// TIA Portal V18 export
FUNCTION_BLOCK "BOOL_DEMUX"   // FB13, LAD
{ S7_Optimized_Access := 'TRUE' }
VERSION : 0.1
// stored: AutoNumber true, IsIECCheckEnabled false, IsRetainMemResEnabled false, MemoryReserve 100, SetENOAutomatically false, UDAEnableTagReadback false
   VAR_INPUT
      State : Int;
      Reset_cmd : Bool;
      Homing_all_axis : Bool;
   END_VAR
   VAR_OUTPUT
      Out1 { ExternalAccessible := 'False'; ExternalVisible := 'False'; ExternalWritable := 'False'} : Bool;
      Out2 { ExternalAccessible := 'False'; ExternalVisible := 'False'; ExternalWritable := 'False'} : Bool;
      Out3 { ExternalAccessible := 'False'; ExternalVisible := 'False'; ExternalWritable := 'False'} : Bool;
      Out4 { ExternalAccessible := 'False'; ExternalVisible := 'False'; ExternalWritable := 'False'} : Bool;
      Out5 { ExternalAccessible := 'False'; ExternalVisible := 'False'; ExternalWritable := 'False'} : Bool;
      Out6 : Int;
   END_VAR
   VAR
      Edge_S_Out1 : Bool;
      Edge_M_Out1 : Bool;
      Edge_S_Out2 : Bool;
      Edge_M_Out2 : Bool;
      Edge_S_Out3 : Bool;
      Edge_M_Out3 : Bool;
      Edge_S_Out4 : Bool;
      Edge_M_Out4 : Bool;
      Edge_S_Out5 : Bool;
      Edge_M_Out5 : Bool;
   END_VAR
   VAR_TEMP   // added for the SCL form of the ladder/FBD networks
      _w1 : Bool;
   END_VAR
BEGIN

REGION Network 1
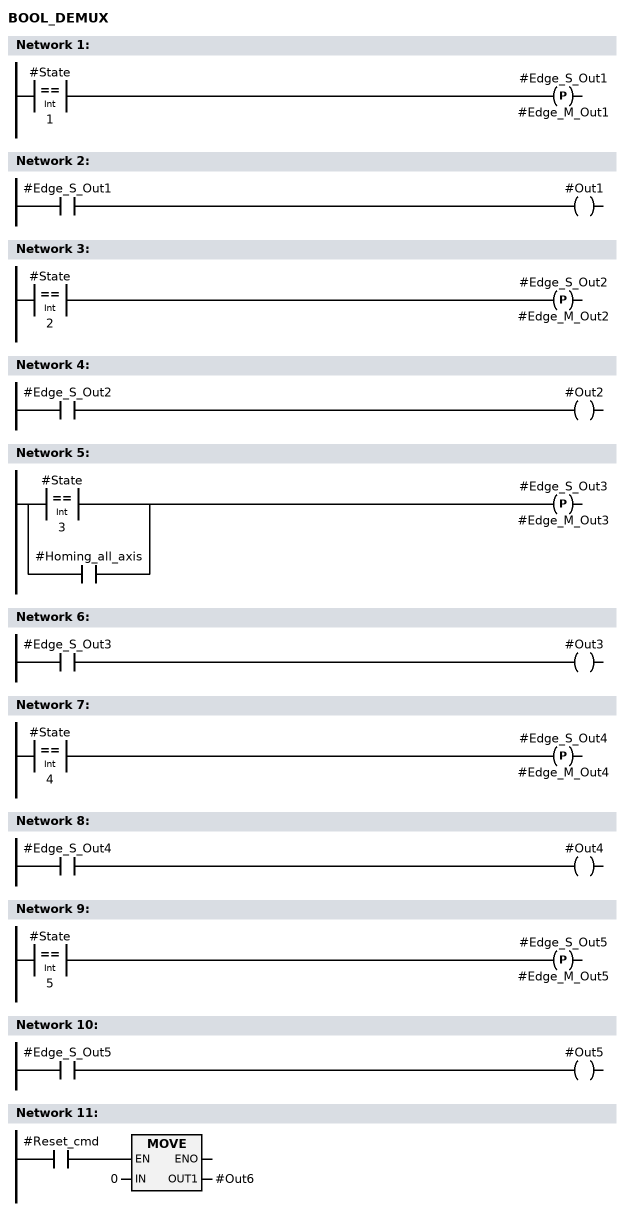
   #_w1 := #State = 1;
   #Edge_S_Out1 := #_w1 AND NOT #Edge_M_Out1;   // rising edge
   #Edge_M_Out1 := #_w1;
END_REGION

REGION Network 2
   RUNG wire#powerrail
      Contact( #Edge_S_Out1 )
      Coil( #Out1 )
   END_RUNG
   // the same network as SCL:
   #Out1 := #Edge_S_Out1;
END_REGION

REGION Network 3
   #_w1 := #State = 2;
   #Edge_S_Out2 := #_w1 AND NOT #Edge_M_Out2;   // rising edge
   #Edge_M_Out2 := #_w1;
END_REGION

REGION Network 4
   RUNG wire#powerrail
      Contact( #Edge_S_Out2 )
      Coil( #Out2 )
   END_RUNG
   // the same network as SCL:
   #Out2 := #Edge_S_Out2;
END_REGION

REGION Network 5
   #_w1 := (#State = 3) OR #Homing_all_axis;
   #Edge_S_Out3 := #_w1 AND NOT #Edge_M_Out3;   // rising edge
   #Edge_M_Out3 := #_w1;
END_REGION

REGION Network 6
   RUNG wire#powerrail
      Contact( #Edge_S_Out3 )
      Coil( #Out3 )
   END_RUNG
   // the same network as SCL:
   #Out3 := #Edge_S_Out3;
END_REGION

REGION Network 7
   #_w1 := #State = 4;
   #Edge_S_Out4 := #_w1 AND NOT #Edge_M_Out4;   // rising edge
   #Edge_M_Out4 := #_w1;
END_REGION

REGION Network 8
   RUNG wire#powerrail
      Contact( #Edge_S_Out4 )
      Coil( #Out4 )
   END_RUNG
   // the same network as SCL:
   #Out4 := #Edge_S_Out4;
END_REGION

REGION Network 9
   #_w1 := #State = 5;
   #Edge_S_Out5 := #_w1 AND NOT #Edge_M_Out5;   // rising edge
   #Edge_M_Out5 := #_w1;
END_REGION

REGION Network 10
   RUNG wire#powerrail
      Contact( #Edge_S_Out5 )
      Coil( #Out5 )
   END_RUNG
   // the same network as SCL:
   #Out5 := #Edge_S_Out5;
END_REGION

REGION Network 11
   RUNG wire#powerrail
      Contact( #Reset_cmd )
      Move(in := 0, out1 => #Out6)
   END_RUNG
   // the same network as SCL:
   IF #Reset_cmd THEN #Out6 := 0; END_IF;
END_REGION
END_FUNCTION_BLOCK
